TYPE McMoveRelativeProcessArgs :
STRUCT
	///Distance to move
	distance: LREAL;
	///Maximum velocity
	maxVelocity: LREAL;
END_STRUCT
END_TYPE

(* stored: Version 1.1.0.1, ProductVersion 3.1.4019.2
   DUT McMoveRelativeProcessArgs: Id {40ba8f4c-af98-41a4-ad6c-f95e05b08c89} *)
